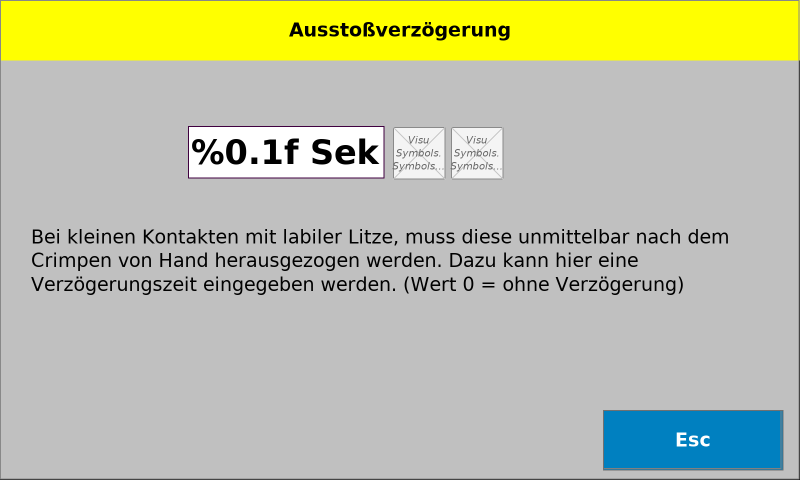
VISUALIZATION Ausstossverz  // 800x480
    Rectangle (0,0 800x480), text variable: DB6.rAusstossverz
    Rectangle (0,0 800x60), "Ausstoßverzögerung"
    Button (603,410 180x60), "Esc"
        OnMouseUp: change screen: Previous 
    Rectangle (188,126 196x52), "%0.1f Sek", text variable: DB6.rAusstossverz
    Image (393,127 52x52), image: VisuSymbols.Symbols.TriangleLeft
        OnMouseClick: execute { P_DecAusstossV(); }
    Image (451,127 52x52), image: VisuSymbols.Symbols.TriangleRight
        OnMouseUp: execute { P_IncAusstossV(); }
    Label (28,224 730x152), "Bei kleinen Kontakten mit labiler Litze, muss diese unmittelbar nach dem Crimpen von Hand herausgezogen werden. Dazu kann hier eine Verzögerungszeit eingegeben werden. (Wert 0 = ohne Verzögerung)"
END_VISUALIZATION

(* stored: Version 1.1.0.1, ProductVersion 3.1.4024.3
   Visu Ausstossverz: Id {f04dbca0-3681-4b35-befa-ef562706adec} *)
